Yaskawa INFORM job: GFG.JBI

/JOB
//NAME GFG
//POS
///NPOS 1,1,0,0,0,0
///TOOL 0
///POSTYPE PULSE
///PULSE
C00000=166224,-110400,-73585,13317,67917,-88284
BC00000=373829,1114849,1075172
//INST
///DATE 2024/01/29 17:50
///ATTR SC,RW
///GROUP1 RB1,BS1
NOP
MOVL C00000 BC00000 V=765.0
END
